# EPICS autosave request: profile_bluesky/startup/ref/Db/USAXSfly_settings.req
#$(P)$(Q)adjustTranLinFrac
$(P)$(Q)AYTolerance
$(P)$(Q)DYTolerance
$(P)$(Q)AYDYstart
file acalcout_settings.req P=$(P)$(Q)acalc1
file acalcout_settings.req P=$(P)$(Q)acalc2
file acalcout_settings.req P=$(P)$(Q)acalc3
file acalcout_settings.req P=$(P)$(Q)acalc4
file acalcout_settings.req P=$(P)$(Q)acalc5
